(* Logix 5000 project; controller TP_EOL20161211 1769-L16ER-BB1B rev 20.12; software revision 20.01 *)

TASK SocketInterface (periodic, rate 100 ms, priority 2, watchdog 500 ms) : Comm

MODULES
   Local : 1769-L16ER-BB1B (PointIO 0, rev 20.12)
      EOL_ENBT_S02 : 1768-ENBT (Ethernet 192.168.1.20, rev 4.1)
         EOL_PLC_S00 : 1768-L43 (1768Ctrl3Slot 0, rev 20.1)
      Discrete_IO : Embedded (PointIO 1, rev 20.11, Output RPI 20 ms)
END_MODULES

TYPE SKT_Addr :
STRUCT
   Family : INT;   // Address Family Must be 2
   Port : INT;   // Port Number
   Addr : SINT[4];   // IP Address
END_STRUCT
END_TYPE

TYPE SKT_CreateParams :
STRUCT
   Type : DINT;   // 1 - TCP 2- UPD
   Addr : SKT_Addr;
END_STRUCT
END_TYPE

TYPE SKT_DATA_CLIENT :
STRUCT
   MSG_Path : STRING;
   Timeout : DINT;
   Create_Source : SKT_CreateParams;
   Instance : DINT;
   Connect_Source : SKT_OpenConnParam;
   Read_Source : SKT_ReadParams;
   Read_Response : SKT_ReadResponse;
   Write_Source : SKT_WriteParams;
   Write_SizeSent : DINT;
END_STRUCT
END_TYPE

TYPE SKT_OpenConnParam :
STRUCT
   Timeout : DINT;
   DestAddr : STRING;
END_STRUCT
END_TYPE

TYPE SKT_ReadParams :
STRUCT
   Timeout : DINT;
   BufLen : DINT;
END_STRUCT
END_TYPE

TYPE SKT_ReadResponse :
STRUCT
   FromAddr : SKT_Addr;
   Buffer : STR_480;
END_STRUCT
END_TYPE

TYPE SKT_WriteParams :
STRUCT
   Timeout : DINT;
   ToAddr : SKT_Addr;
   Buffer : STR_480;
END_STRUCT
END_TYPE

TYPE STR_480 :
STRUCT
   LEN : DINT;
   DATA : SINT[480];
END_STRUCT
END_TYPE

TYPE UDT_EOLPlus :
STRUCT
   String : STRING[25];
   DINT : DINT[10];
   Real : REAL[10];
END_STRUCT
END_TYPE

ADD_ON_INSTRUCTION SKT_TCP_CLIENT_AOI   (* revision 1.0, ExecutePrescan *)
VAR_IN_OUT
   Client_Data : SKT_DATA_CLIENT; {required}   // This tags holds all the data used by the messages
END_VAR
VAR_INPUT
   Enable_Socket : BOOL; {visible}   // Set by user to enable or disable socket
   Stop_On_Error : BOOL; {visible}   // If any message errors, then delete socket and stop
END_VAR
VAR_IN_OUT
   Create_MSG : MESSAGE; {required}   // Create socket
   Connect_MSG : MESSAGE; {required}   // Connect socket to server.
   Read_MSG : MESSAGE; {required}   // Message to tell socket to return any data it has recieved
   Write_MSG : MESSAGE; {required}   // Write socket message
   Delete_MSG : MESSAGE; {required}   // Delete socket
END_VAR
VAR_OUTPUT
   SC : BOOL; {access Read Only, visible}   // Trying to connect to Server.
   SO : BOOL; {access Read Only, visible}   // Socket connection Open
   DR : BOOL; {access Read Only, visible}   // New Data Ready - Set by AOI when a string is received, cleared by user to acknowledge
   WD : BOOL; {access Read Only, visible}   // Set this bit to Write Data
   ER : BOOL; {access Read Only, visible}   // A message had an ERror
END_VAR
VAR
   State : DINT;   // Current state
END_VAR

ROUTINE Logic   (* ladder *)
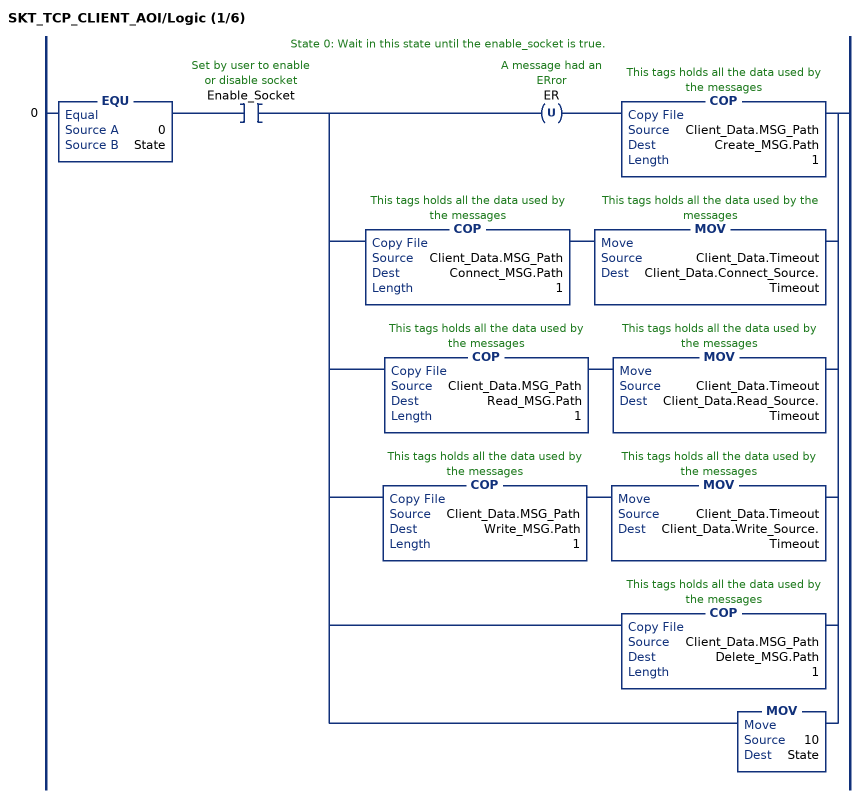
   // State 0: Wait in this state until the enable_socket is true.
   0: EQU(0,State)XIC(Enable_Socket)[OTU(ER) COP(Client_Data.MSG_Path,Create_MSG.Path,1) ,COP(Client_Data.MSG_Path,Connect_MSG.Path,1) MOV(Client_Data.Timeout,Client_Data.Connect_Source.Timeout) ,COP(Client_Data.MSG_Path,Read_MSG.Path,1) MOV(Client_Data.Timeout,Client_Data.Read_Source.Timeout) ,COP(Client_Data.MSG_Path,Write_MSG.Path,1) MOV(Client_Data.Timeout,Client_Data.Write_Source.Timeout) ,COP(Client_Data.MSG_Path,Delete_MSG.Path,1) ,MOV(10,State) ];
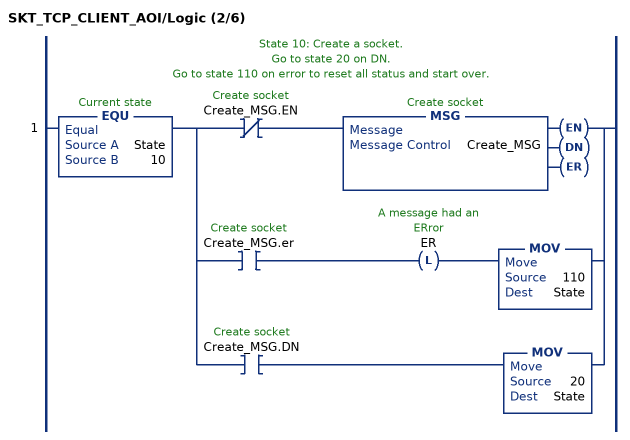
   // State 10: Create a socket.
   // Go to state 20 on DN.
   // Go to state 110 on error to reset all status and start over.
   1: EQU(State,10)[XIO(Create_MSG.EN) MSG(Create_MSG) ,XIC(Create_MSG.er) OTL(ER) MOV(110,State) ,XIC(Create_MSG.DN) MOV(20,State) ];
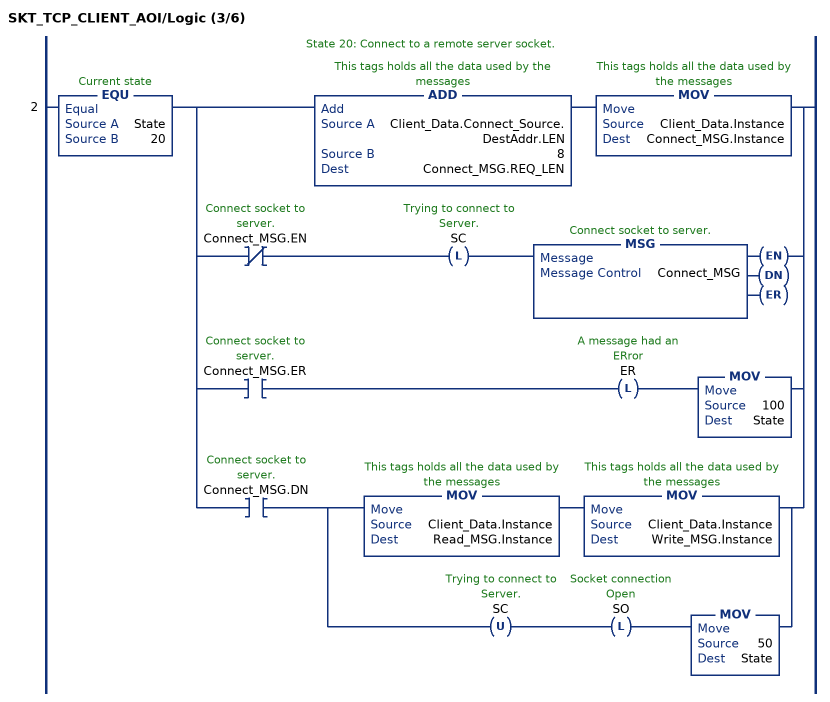
   // State 20: Connect to a remote server socket.
   2: EQU(State,20)[ADD(Client_Data.Connect_Source.DestAddr.LEN,8,Connect_MSG.REQ_LEN) MOV(Client_Data.Instance,Connect_MSG.Instance) ,XIO(Connect_MSG.EN) OTL(SC) MSG(Connect_MSG) ,XIC(Connect_MSG.ER) OTL(ER) MOV(100,State) ,XIC(Connect_MSG.DN) [MOV(Client_Data.Instance,Read_MSG.Instance) MOV(Client_Data.Instance,Write_MSG.Instance) ,OTU(SC) OTL(SO) MOV(50,State) ] ];
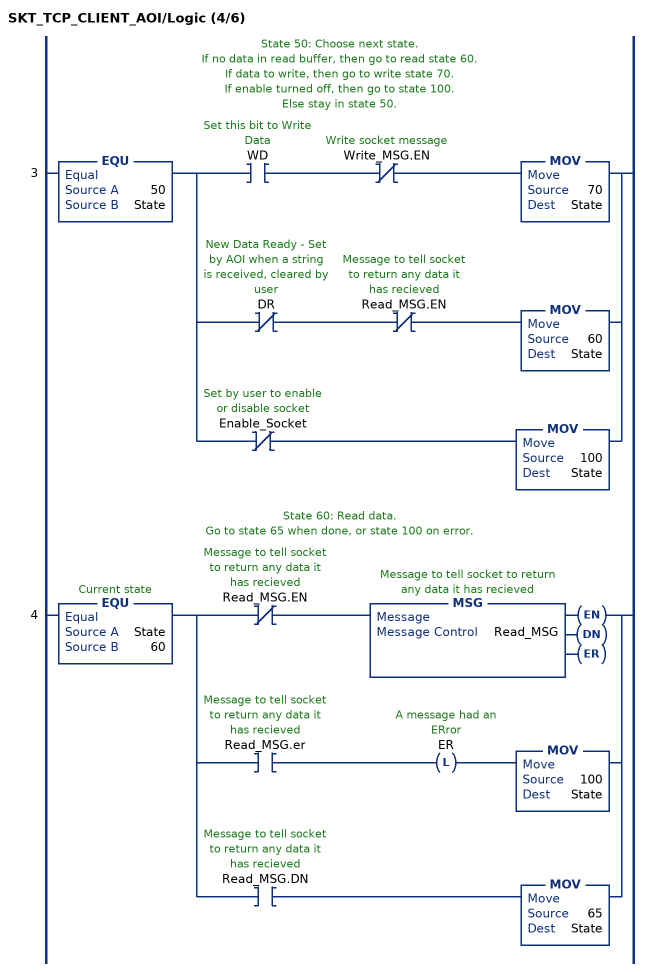
   // State 50: Choose next state.
   // If no data in read buffer, then go to read state 60.
   // If data to write, then go to write state 70.
   // If enable turned off, then go to state 100.
   // Else stay in state 50.
   3: EQU(50,State)[XIC(WD) XIO(Write_MSG.EN) MOV(70,State) ,XIO(DR) XIO(Read_MSG.EN) MOV(60,State) ,XIO(Enable_Socket) MOV(100,State) ];
   // State 60: Read data.
   // Go to state 65 when done, or state 100 on error.
   4: EQU(State,60)[XIO(Read_MSG.EN) MSG(Read_MSG) ,XIC(Read_MSG.er) OTL(ER) MOV(100,State) ,XIC(Read_MSG.DN) MOV(65,State) ];
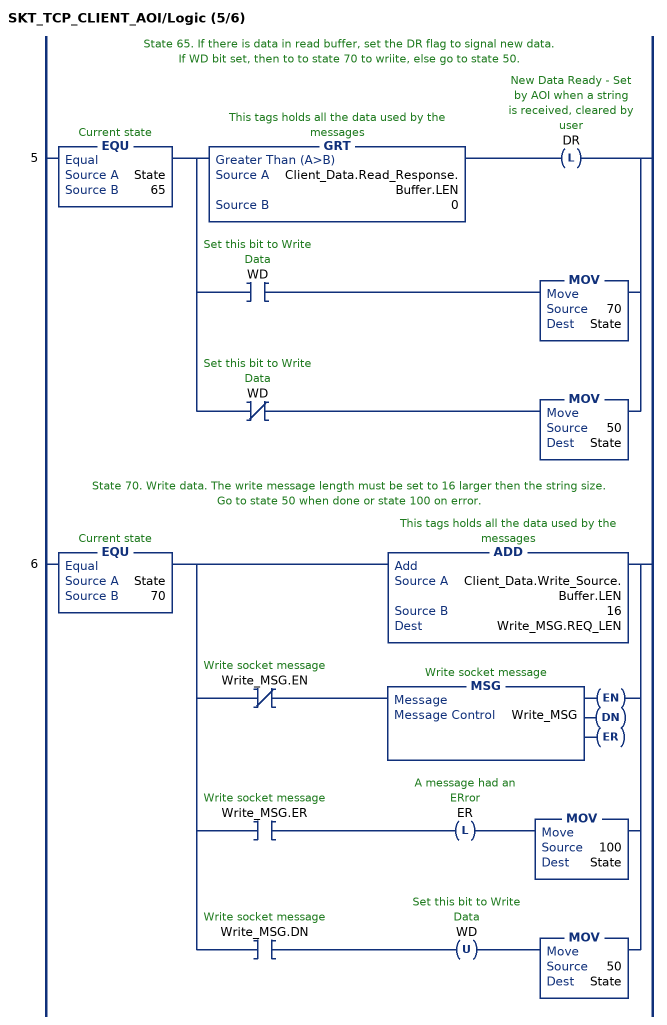
   // State 65. If there is data in read buffer, set the DR flag to signal new data.
   // If WD bit set, then to to state 70 to wriite, else go to state 50.
   5: EQU(State,65)[GRT(Client_Data.Read_Response.Buffer.LEN,0) OTL(DR) ,XIC(WD) MOV(70,State) ,XIO(WD) MOV(50,State) ];
   // State 70. Write data. The write message length must be set to 16 larger then the string size.
   // Go to state 50 when done or state 100 on error.
   6: EQU(State,70)[ADD(Client_Data.Write_Source.Buffer.LEN,16,Write_MSG.REQ_LEN) ,XIO(Write_MSG.EN) MSG(Write_MSG) ,XIC(Write_MSG.ER) OTL(ER) MOV(100,State) ,XIC(Write_MSG.DN) OTU(WD) MOV(50,State) ];
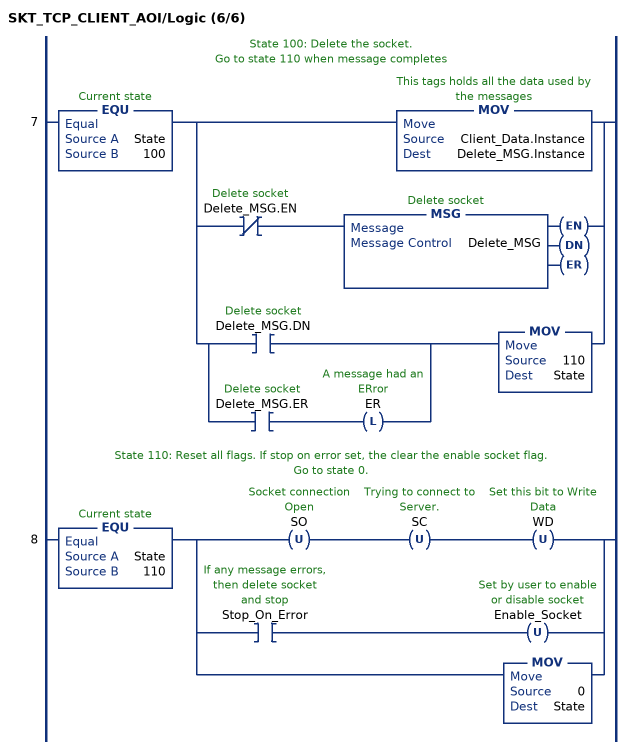
   // State 100: Delete the socket.
   // Go to state 110 when message completes
   7: EQU(State,100)[MOV(Client_Data.Instance,Delete_MSG.Instance) ,XIO(Delete_MSG.EN) MSG(Delete_MSG) ,[XIC(Delete_MSG.DN) ,XIC(Delete_MSG.ER) OTL(ER) ] MOV(110,State) ];
   // State 110: Reset all flags. If stop on error set, the clear the enable socket flag.
   // Go to state 0.
   8: EQU(State,110)[OTU(SO) OTU(SC) OTU(WD) ,XIC(Stop_On_Error) OTU(Enable_Socket) ,MOV(0,State) ];
END_ROUTINE

ROUTINE Prescan   (* ladder *)
// Prescan
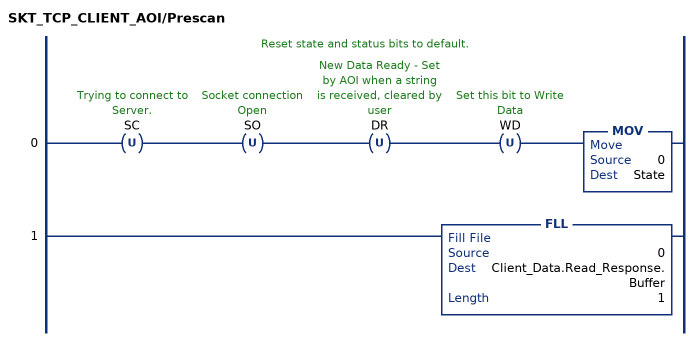
   // Reset state and status bits to default.
   0: OTU(SC)OTU(SO)OTU(DR)OTU(WD)MOV(0,State);
   1: FLL(0,Client_Data.Read_Response.Buffer,1);
END_ROUTINE
END_ADD_ON_INSTRUCTION

VAR_GLOBAL   (* controller tags *)
   ACW_CO_Step : INT;
   ACW_SKT_Client_Connect_MSG : MESSAGE;
        MessageParameters(ServiceCode := 16#004c, LocalElement := ACW_SKT_Client_DATA.Connect_Source, ...)
   ACW_SKT_Client_Create_MSG : MESSAGE;
        MessageParameters(ServiceCode := 16#004b, LocalElement := ACW_SKT_Client_DATA.Create_Source, DestinationTag := ACW_SKT_Client_DATA.Instance, ...)
   ACW_SKT_Client_DATA : SKT_DATA_CLIENT := (MSG_Path := '$01$00', Timeout := 2000, Create_Source.Type := 1, Create_Source.Addr.Family := 2, Instance := 27231, Connect_Source.Timeout := 2000, Connect_Source.DestAddr := '192.168.1.68?port=50001', Read_Source.Timeout := 2000, Read_Source.BufLen := 480, Read_Response.Buffer := '$0233991118247.001$03', Write_Source.Timeout := 2000, Write_Source.ToAddr.Family := 2, Write_Source.Buffer := '$02339$03', Write_SizeSent := 5);
   ACW_SKT_Client_Delete_MSG : MESSAGE;
        MessageParameters(ServiceCode := 16#004f, ...)
   ACW_SKT_Client_Port : DINT;
   ACW_SKT_Client_Read_MSG : MESSAGE;
        MessageParameters(ServiceCode := 16#004d, LocalElement := ACW_SKT_Client_DATA.Read_Source, DestinationTag := ACW_SKT_Client_DATA.Read_Response, ...)
   ACW_SKT_Client_Write_MSG : MESSAGE;
        MessageParameters(ServiceCode := 16#004e, LocalElement := ACW_SKT_Client_DATA.Write_Source, DestinationTag := ACW_SKT_Client_DATA.Write_SizeSent, ...)
   ACW_SKT_Delete_All_MSG : MESSAGE;
        MessageParameters(ServiceCode := 16#0051, ...)
   ACW_SKT_Device_IP_Port_Server : STRING := '192.168.1.68?port=50001';
   ACW_SKT_MSG_PATH : STRING := '$01$00';
   ACW_SKT_String_recieved : STR_480 := '$020100000100$03';
   ACW_SKT_String_to_send : STR_480 := '$02339$03';
   ACW_SKT_Toggle : DINT := -2147482592;
        .0   // Toggle to delete all sockets
   EOL_MSGRead : MESSAGE;
        MessageParameters(ServiceCode := 16#004c, LocalElement := nc_CO_Cmd, ...)
   EOL_MSGWrite : MESSAGE;
        MessageParameters(ServiceCode := 16#004d, LocalElement := np_CO_Status, ...)
   nc_CO_Cmd : UDT_EOLPlus := (String[2] := '5177', String[3] := '457', String[4] := '84', DINT[0] := 2);
   nc_COData : UDT_EOLPlus;
   nc_COData_String : STRING[25];
   np_CO_Status : UDT_EOLPlus := (DINT[0] := 1);
   SKT_Delete_All_MSG : MESSAGE;
        MessageParameters(ServiceCode := 16#0051, ...)
   VDS_SKT_Client_Connect_MSG : MESSAGE;
        MessageParameters(ServiceCode := 16#004c, LocalElement := VDS_SKT_Client_DATA.Connect_Source, ...)
   VDS_SKT_Client_Create_MSG : MESSAGE;
        MessageParameters(ServiceCode := 16#004b, LocalElement := VDS_SKT_Client_DATA.Create_Source, DestinationTag := VDS_SKT_Client_DATA.Instance, ...)
   VDS_SKT_Client_DATA : SKT_DATA_CLIENT := (MSG_Path := '$01$00', Timeout := 2000, Create_Source.Type := 1, Create_Source.Addr.Family := 2, Instance := 19462, Connect_Source.Timeout := 2000, Connect_Source.DestAddr := '192.168.1.66?port=3004', Read_Source.Timeout := 2000, Read_Source.BufLen := 480, Write_Source.Timeout := 2000, Write_Source.ToAddr.Family := 2, Write_Source.Buffer := 'SEL|82254066|$0D', Write_SizeSent := 14);
   VDS_SKT_Client_Delete_MSG : MESSAGE;
        MessageParameters(ServiceCode := 16#004f, ...)
   VDS_SKT_Client_Port : DINT;
   VDS_SKT_Client_Read_MSG : MESSAGE;
        MessageParameters(ServiceCode := 16#004d, LocalElement := VDS_SKT_Client_DATA.Read_Source, DestinationTag := VDS_SKT_Client_DATA.Read_Response, ...)
   VDS_SKT_Client_Write_MSG : MESSAGE;
        MessageParameters(ServiceCode := 16#004e, LocalElement := VDS_SKT_Client_DATA.Write_Source, DestinationTag := VDS_SKT_Client_DATA.Write_SizeSent, ...)
   VDS_SKT_Delete_All_MSG : MESSAGE;
        MessageParameters(ServiceCode := 16#0051, ...)
   VDS_SKT_Device_IP_Port_Server : STRING := '192.168.1.66?port=3004';
   VDS_SKT_MSG_PATH : STRING := '$01$00';
   VDS_SKT_String_recieved : STR_480 := 'ACK$0D';
   VDS_SKT_String_to_send : STR_480 := 'SEL|82254066|$0D';
   VDS_SKT_Toggle : DINT := 1056;
        .0   // Toggle to delete all sockets
   VOS_SKT_Client_Connect_MSG : MESSAGE;
        MessageParameters(ServiceCode := 16#004c, LocalElement := VOS_SKT_Client_DATA.Connect_Source, ...)
   VOS_SKT_Client_Create_MSG : MESSAGE;
        MessageParameters(ServiceCode := 16#004b, LocalElement := VOS_SKT_Client_DATA.Create_Source, DestinationTag := VOS_SKT_Client_DATA.Instance, ...)
   VOS_SKT_Client_DATA : SKT_DATA_CLIENT := (MSG_Path := '$01$00', Timeout := 2000, Create_Source.Type := 1, Create_Source.Addr.Family := 2, Instance := 26707, Connect_Source.Timeout := 2000, Connect_Source.DestAddr := '192.168.1.65?port=3003', Read_Source.Timeout := 2000, Read_Source.BufLen := 480, Write_Source.Timeout := 2000, Write_Source.ToAddr.Family := 2, Write_Source.Buffer := 'SLA|82254066|PLC01=6455B002A4|$0D', Write_SizeSent := 31);
   VOS_SKT_Client_Delete_MSG : MESSAGE;
        MessageParameters(ServiceCode := 16#004f, ...)
   VOS_SKT_Client_Port : DINT;
   VOS_SKT_Client_Read_MSG : MESSAGE;
        MessageParameters(ServiceCode := 16#004d, LocalElement := VOS_SKT_Client_DATA.Read_Source, DestinationTag := VOS_SKT_Client_DATA.Read_Response, ...)
   VOS_SKT_Client_Write_MSG : MESSAGE;
        MessageParameters(ServiceCode := 16#004e, LocalElement := VOS_SKT_Client_DATA.Write_Source, DestinationTag := VOS_SKT_Client_DATA.Write_SizeSent, ...)
   VOS_SKT_Delete_All_MSG : MESSAGE;
        MessageParameters(ServiceCode := 16#0051, ...)
   VOS_SKT_Device_IP_Port_Server : STRING := '192.168.1.65?port=3003';
   VOS_SKT_MSG_PATH : STRING := '$01$00';
   VOS_SKT_String_recieved : STR_480 := 'JDL|6|Copy of Field00=82254066|Copy of Field02=HAIR FALL CONTROL|Copy of Field04=10:06|Copy of Field03=14902430400883|Copy of Field01=|PLC01=6455B002A4|$0D';
   VOS_SKT_String_to_send : STR_480 := 'GJN$0D';
   VOS_SKT_Toggle : DINT := 1056;
        .0   // Toggle to delete all sockets
   wrk_Ons : INT := 512;
END_VAR

PROGRAM Comm   (* main routine Main *)
VAR
   aa_Dint : DINT := 2;
   aa_FSC : CONTROL := (LEN := 20, POS := 9, EN := 1, IN := 1, FD := 1);
   aa_STD : CONTROL := (LEN := 20);
   aa_STD1 : CONTROL := (LEN := 6);
   ACW_Add : DINT;
   ACW_Cmd_ConvStart : BOOL;
   ACW_Cmd_ConvStop : BOOL := 1;
   ACW_CO_Timer : TIMER[10] := ([0].PRE := 1000);
   acw_ConvStopped : STRING := '$020100000100$03';
   ACW_SKT_Client_AOI : SKT_TCP_CLIENT_AOI := (Enable_Socket := 1, SO := 1, DR := 1);
   Araa : CONTROL := (LEN := 20, POS := 17);
   Array : REAL[20] := ([6] := 2.0, [7] := 15.0, [8] := 45.0, [9] := 54.0, [10] := 54.0, [11] := 55.0, [12] := 55.0, [13] := 55.3, [14] := 56.0, [15] := 56.2, [16] := 56.5, [17] := 57.0, [18] := 57.8, [19] := 65.0);
   Array2 : REAL[20];
   Cmd_ACW_ConvStart : STRING := '$0212$03'; {constant}
   Cmd_ACW_ConvStop : STRING := '$02339$03'; {constant}
   Cmd_ACW_RecipeName : STRING := '91118247.001';
   Cmd_ACW_RecipeNumber : STRING := '$0220001$03';
   Cmd_ACW_SetRecipeName : BOOL;
   Cmd_ACW_SetRecipeNumber : BOOL;
   Cmd_ACW_SetTargetLL : BOOL;
   Cmd_ACW_SetTargetUL : BOOL;
   Cmd_ACW_SetTargetWeight : BOOL;
   Cmd_ACW_Status : STRING;
   Cmd_ACW_TargetLL : STRING := '84';
   Cmd_ACW_TargetUL : STRING := '457';
   Cmd_ACW_TargetWeight : STRING := '5177';
   Cmd_Chk : INT;
   Cmd_RecipeNo : BOOL;
   Cmd_RequestData : STRING := '$020$03'; {constant}
   Cmd_VJDS_GJD : BOOL;
   Cmd_VJDS_GJF : BOOL;
   Cmd_VJDS_GJN : BOOL;
   Cmd_VJDS_GST : BOOL;
   Cmd_VJDS_OfflineRequest : BOOL;
   Cmd_VJDS_RunRequest : BOOL;
   Cmd_VJDS_SEL : BOOL;
   Cmd_VJDS_ShutDownRequest : BOOL;
   Cmd_VJDS_ShuttingDownRequest : BOOL;
   Cmd_VJDS_SLA : BOOL;
   Cmd_VJDS_StartupRequest : BOOL;
   Cmd_VJOS_GJD : BOOL;
   Cmd_VJOS_GJF : BOOL;
   Cmd_VJOS_GJN : BOOL;
   Cmd_VJOS_GST : BOOL;
   Cmd_VJOS_OfflineRequest : BOOL;
   Cmd_VJOS_RunRequest : BOOL;
   Cmd_VJOS_ShutDownRequest : BOOL;
   Cmd_VJOS_ShuttingDownRequest : BOOL;
   Cmd_VJOS_SLA : BOOL;
   Cmd_VJOS_StartupRequest : BOOL;
   CO_Complete : TIMER := (PRE := 180000);
   CO_Trigger : DINT := 6;
   CO_VJCTU : COUNTER := (ACC := 2, CU := 1, DN := 1);
   CO_VJCTUOS : COUNTER := (ACC := 2, CU := 1, DN := 1);
   FSC : CONTROL;
   Par_JobSelect : STRING := '82254066';
   Par_RecipeName : STRING := '$02239$03';
   Par_TargetLL : STRING := '$02203-$03';
   Par_TargetUL : STRING := '$02202$03';
   Par_TargetWeight : STRING := '$02201$03';
   Par_VarData : STRING := '6455B002A4';
   Par_VJ_JobSelect : STRING := '82254066';
   RCO_Triggered : INT := 4;
   Real_STD : REAL := 27.257544;
   Sts_Conv : STRING := '1';
   Sts_VJDS_CurrentJob : STRING;
   Sts_VJOS_CurrentJob : STRING := '82254066';
   VDS_SKT_Client_AOI : SKT_TCP_CLIENT_AOI := (Enable_Socket := 1, SO := 1);
   VJ_ACK : STRING := 'ACK$0D';
   VJ_Blank : STRING;
   VJ_FieldData : STRING := '6455B002A4';
   VJ_FieldDataDS : STRING;
   VJ_FieldPos : INT := 136;
   VJ_FieldPosDS : INT;
   VJ_PLC01 : STRING := 'PLC01='; {constant}
   VJ_VarDataPOS : INT := 142;
   VJDS_JobFieldDataErr : BOOL;
   VJDS_JobFieldDataNA : BOOL;
   VJDS_JobSLAErr : BOOL;
   VJDS_msgSeq : INT := 60;
   VJDS_ReadTimer : TIMER[10] := ([0].PRE := 2000, [1].PRE := 2000, [2].PRE := 2000, [3].PRE := 2000, [3].ACC := 2000, [3].EN := 1, [3].DN := 1, [4].PRE := 2000, [5].PRE := 2000, [6].PRE := 3000);
   VJDS_Wrk_Jobassign : STRING := '82254066|PLC01=6455B002A4';
   VJDS_wrk_ONS : DINT;
   VJOS_JobFieldDataErr : BOOL;
   VJOS_JobSLAErr : BOOL;
   VJOS_msgSeq : INT := 30;
   VJOS_ReadTimer : TIMER[10] := ([0].PRE := 2000, [1].PRE := 2000, [2].PRE := 2000, [2].ACC := 2000, [2].EN := 1, [2].DN := 1, [3].PRE := 2000, [4].PRE := 2000, [5].PRE := 2000, [6].PRE := 3000);
   VJOS_Seq : INT := 10;
   VJOS_Wrk_Jobassign : STRING := '82254066|PLC01=6455B002A4';
   VJOS_wrk_ONS : DINT := 32;
   VOS_SKT_Client_AOI : SKT_TCP_CLIENT_AOI := (Enable_Socket := 1, SO := 1);
   wrk_Concat : STRING := '82254066|PLC01=';
   wrk_ConcatSLA : STRING := '|PLC01='; {constant}
   wrk_GJD : STRING := 'GJD$0D'; {constant}
   wrk_GJF : STRING := 'GJF||$0D'; {constant}
   wrk_GJN : STRING := 'GJN$0D'; {constant}
   wrk_GST : STRING := 'GST$0D'; {constant}
   wrk_SEL : STRING := 'SEL||$0D'; {constant}
   wrk_SLA : STRING := 'SLA||$0D'; {constant}
   wrk_State : STRING := '3';
   wrk_StateCmd : STRING := 'SST||$0D'; {constant}
END_VAR

ROUTINE Anritsu   (* ladder *)
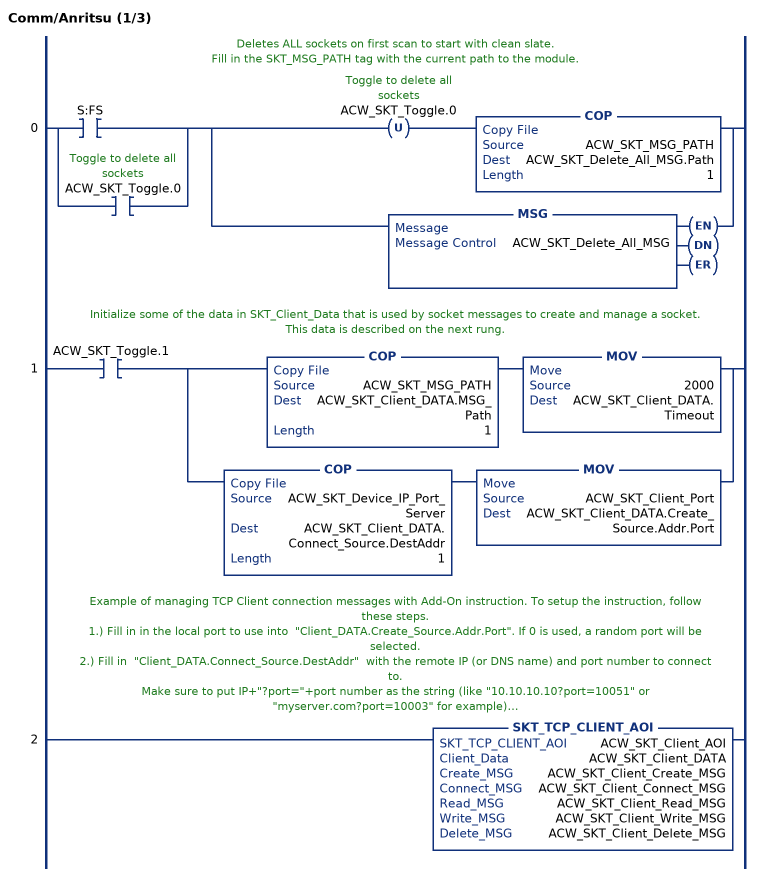
   // Deletes ALL sockets on first scan to start with clean slate.
   // Fill in the SKT_MSG_PATH tag with the current path to the module.
   0: [XIC(S:FS) ,XIC(ACW_SKT_Toggle.0) ][OTU(ACW_SKT_Toggle.0) COP(ACW_SKT_MSG_PATH,ACW_SKT_Delete_All_MSG.Path,1) ,MSG(ACW_SKT_Delete_All_MSG) ];
   // Initialize some of the data in SKT_Client_Data that is used by socket messages to create and manage a socket.
   // This data is described on the next rung.
   1: XIC(ACW_SKT_Toggle.1)[COP(ACW_SKT_MSG_PATH,ACW_SKT_Client_DATA.MSG_Path,1) MOV(2000,ACW_SKT_Client_DATA.Timeout) ,COP(ACW_SKT_Device_IP_Port_Server,ACW_SKT_Client_DATA.Connect_Source.DestAddr,1) MOV(ACW_SKT_Client_Port,ACW_SKT_Client_DATA.Create_Source.Addr.Port) ];
   // Example of managing TCP Client connection messages with Add-On instruction. To setup the instruction, follow these steps.
   // 1.) Fill in in the local port to use into  "Client_DATA.Create_Source.Addr.Port". If 0 is used, a random port will be selected.
   // 2.) Fill in  "Client_DATA.Connect_Source.DestAddr"  with the remote IP (or DNS name) and port number to connect to.
   // Make sure to put IP+"?port="+port number as the string (like "10.10.10.10?port=10051" or "myserver.com?port=10003" for example).
   // 3.) Fill in the path to the module in the SKT_MSG_PATH tag (the path will look like "$01$03" for slot 3, for example).
   // 4.) To start or stop the client connection, set or clear the Enable_Socket respectively.
   // 5.) If trying to trap error for troubleshooting the connection, the set the Stop_on_Error bit on the instruction. If there is an error, the instruction will clear the Stop_on_Errorwhen a message errors.
   // The SC status bit means trying to connect. The SO status bit means Socket Connected and open. The ER bit means a message ERrored.
   // When the DR bit is set by the instruction, then there is string data that arrived from the socket. Copy the string data if desired and clear the DR bit to get new data.
   // When data needs to be sent by the application, fill in the string data into "Client_DATA.Write_Source.Buffer", then set the WD bit. The instruction will clear the WD bit when the data is written.
   // Modify the rung branches to suit the application.
   2: SKT_TCP_CLIENT_AOI(ACW_SKT_Client_AOI,ACW_SKT_Client_DATA,ACW_SKT_Client_Create_MSG,ACW_SKT_Client_Connect_MSG,ACW_SKT_Client_Read_MSG,ACW_SKT_Client_Write_MSG,ACW_SKT_Client_Delete_MSG);
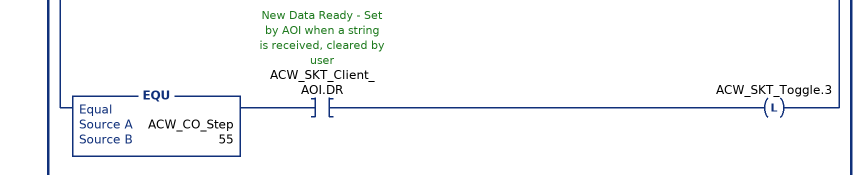
   3: [EQU(ACW_CO_Step,0) [XIC(ACW_Cmd_ConvStart) ONS(wrk_Ons.8) COP(Cmd_ACW_ConvStart,ACW_SKT_String_to_send,Cmd_ACW_ConvStart.LEN) ,XIC(ACW_Cmd_ConvStop) ONS(wrk_Ons.9) COP(Cmd_ACW_ConvStop,ACW_SKT_String_to_send,Cmd_ACW_ConvStop.LEN) ] OTL(ACW_SKT_Toggle.2) ,XIC(nc_CO_Cmd.DINT[0].2) ONS(wrk_Ons.1) MOV(10,ACW_CO_Step) ,XIO(ACW_CO_Timer[0].DN) LIM(10,ACW_CO_Step,60) TON(ACW_CO_Timer[0],?,?) ,XIC(ACW_CO_Timer[0].DN) ADD(ACW_CO_Step,5,ACW_CO_Step) ,EQU(ACW_CO_Step,10) XIO(ACW_SKT_Client_AOI.WD) COP(Cmd_ACW_RecipeNumber,ACW_SKT_String_to_send,Cmd_ACW_RecipeNumber.LEN) OTL(ACW_SKT_Toggle.2) ,EQU(ACW_CO_Step,15) XIC(ACW_SKT_Client_AOI.DR) OTL(ACW_SKT_Toggle.3) ,EQU(ACW_CO_Step,20) XIO(ACW_SKT_Client_AOI.WD) INSERT(Par_RecipeName,Cmd_ACW_RecipeName,5,ACW_SKT_String_to_send) OTL(ACW_SKT_Toggle.2) ,EQU(ACW_CO_Step,25) XIC(ACW_SKT_Client_AOI.DR) OTL(ACW_SKT_Toggle.3) ,EQU(ACW_CO_Step,30) XIO(ACW_SKT_Client_AOI.WD) INSERT(Par_TargetWeight,Cmd_ACW_TargetWeight,5,ACW_SKT_String_to_send) OTL(ACW_SKT_Toggle.2) ,EQU(ACW_CO_Step,35) XIC(ACW_SKT_Client_AOI.DR) OTL(ACW_SKT_Toggle.3) ,EQU(ACW_CO_Step,40) XIO(ACW_SKT_Client_AOI.WD) INSERT(Par_TargetUL,Cmd_ACW_TargetUL,5,ACW_SKT_String_to_send) OTL(ACW_SKT_Toggle.2) ,EQU(ACW_CO_Step,45) XIC(ACW_SKT_Client_AOI.DR) OTL(ACW_SKT_Toggle.3) ,EQU(ACW_CO_Step,50) XIO(ACW_SKT_Client_AOI.WD) INSERT(Par_TargetLL,Cmd_ACW_TargetLL,6,ACW_SKT_String_to_send) OTL(ACW_SKT_Toggle.2) ,EQU(ACW_CO_Step,55) XIC(ACW_SKT_Client_AOI.DR) OTL(ACW_SKT_Toggle.3) ];
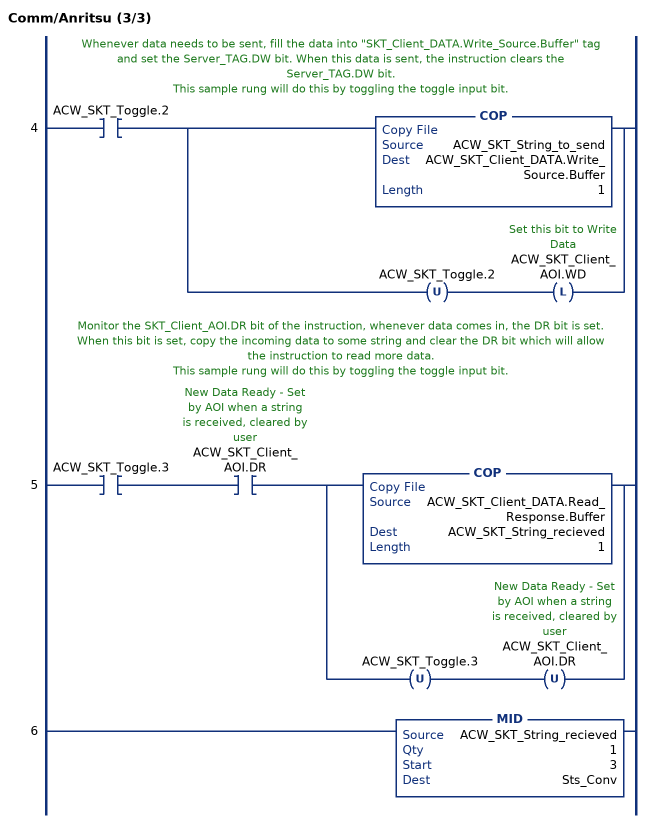
   // Whenever data needs to be sent, fill the data into "SKT_Client_DATA.Write_Source.Buffer" tag and set the Server_TAG.DW bit. When this data is sent, the instruction clears the Server_TAG.DW bit.
   // This sample rung will do this by toggling the toggle input bit.
   4: XIC(ACW_SKT_Toggle.2)[COP(ACW_SKT_String_to_send,ACW_SKT_Client_DATA.Write_Source.Buffer,1) ,OTU(ACW_SKT_Toggle.2) OTL(ACW_SKT_Client_AOI.WD) ];
   // Monitor the SKT_Client_AOI.DR bit of the instruction, whenever data comes in, the DR bit is set. When this bit is set, copy the incoming data to some string and clear the DR bit which will allow the instruction to read more data.
   // This sample rung will do this by toggling the toggle input bit.
   5: XIC(ACW_SKT_Toggle.3)XIC(ACW_SKT_Client_AOI.DR)[COP(ACW_SKT_Client_DATA.Read_Response.Buffer,ACW_SKT_String_recieved,1) ,OTU(ACW_SKT_Toggle.3) OTU(ACW_SKT_Client_AOI.DR) ];
   6: MID(ACW_SKT_String_recieved,1,3,Sts_Conv);
END_ROUTINE

ROUTINE Main   (* ladder *)
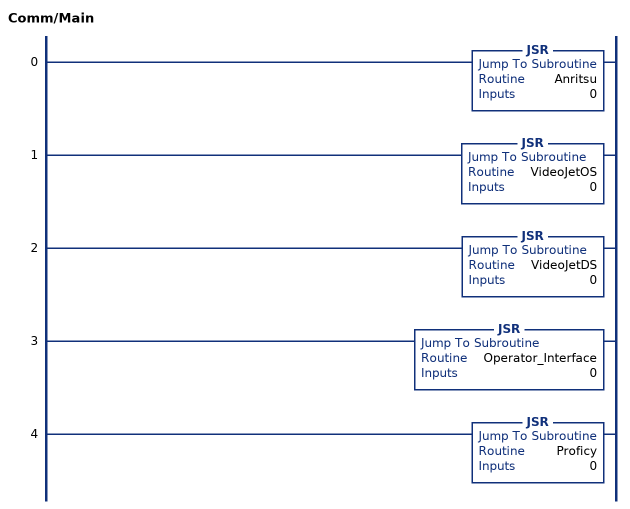
   0: JSR(Anritsu,0);
   1: JSR(VideoJetOS,0);
   2: JSR(VideoJetDS,0);
   3: JSR(Operator_Interface,0);
   4: JSR(Proficy,0);
END_ROUTINE

ROUTINE Operator_Interface   (* ladder *)
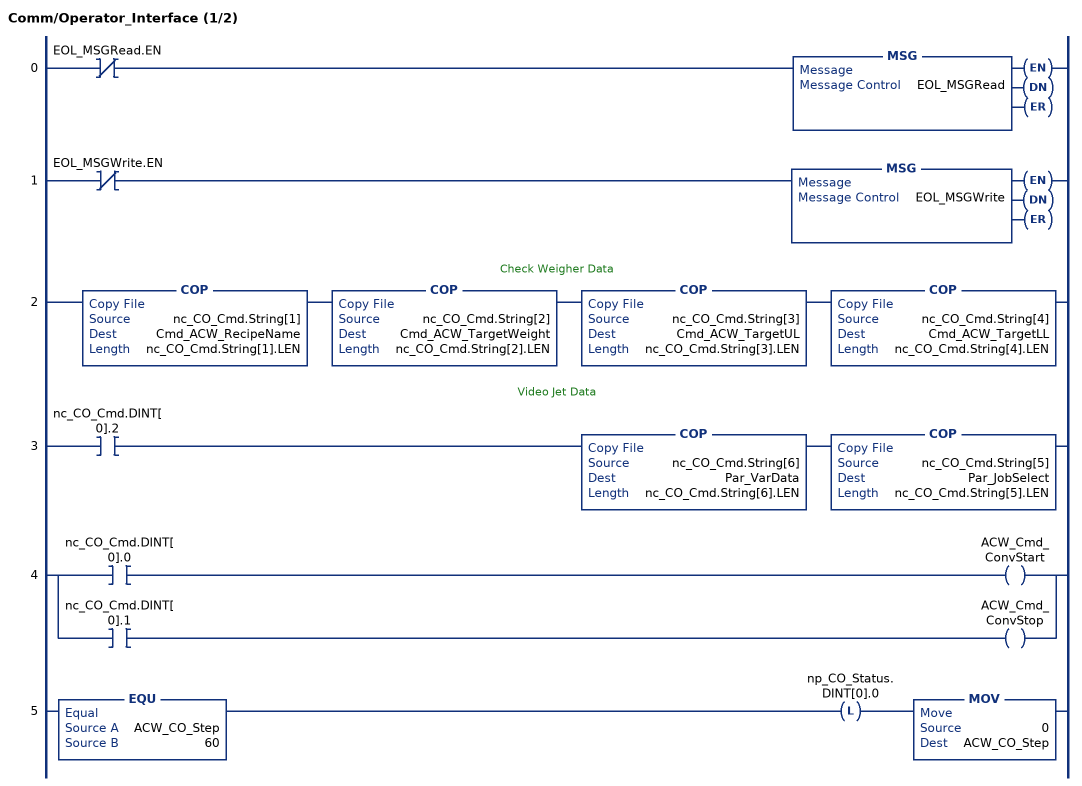
   0: XIO(EOL_MSGRead.EN)MSG(EOL_MSGRead);
   1: XIO(EOL_MSGWrite.EN)MSG(EOL_MSGWrite);
   // Check Weigher Data
   2: COP(nc_CO_Cmd.String[1],Cmd_ACW_RecipeName,nc_CO_Cmd.String[1].LEN)COP(nc_CO_Cmd.String[2],Cmd_ACW_TargetWeight,nc_CO_Cmd.String[2].LEN)COP(nc_CO_Cmd.String[3],Cmd_ACW_TargetUL,nc_CO_Cmd.String[3].LEN)COP(nc_CO_Cmd.String[4],Cmd_ACW_TargetLL,nc_CO_Cmd.String[4].LEN);
   // Video Jet Data
   3: XIC(nc_CO_Cmd.DINT[0].2)COP(nc_CO_Cmd.String[6],Par_VarData,nc_CO_Cmd.String[6].LEN)COP(nc_CO_Cmd.String[5],Par_JobSelect,nc_CO_Cmd.String[5].LEN);
   4: [XIC(nc_CO_Cmd.DINT[0].0) OTE(ACW_Cmd_ConvStart) ,XIC(nc_CO_Cmd.DINT[0].1) OTE(ACW_Cmd_ConvStop) ];
   5: EQU(ACW_CO_Step,60)OTL(np_CO_Status.DINT[0].0)MOV(0,ACW_CO_Step);
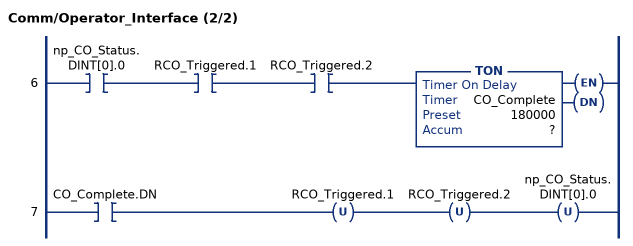
   6: XIC(np_CO_Status.DINT[0].0)XIC(RCO_Triggered.1)XIC(RCO_Triggered.2)TON(CO_Complete,?,?);
   7: XIC(CO_Complete.DN)OTU(RCO_Triggered.1)OTU(RCO_Triggered.2)OTU(np_CO_Status.DINT[0].0);
END_ROUTINE

ROUTINE Proficy   (* ladder *)
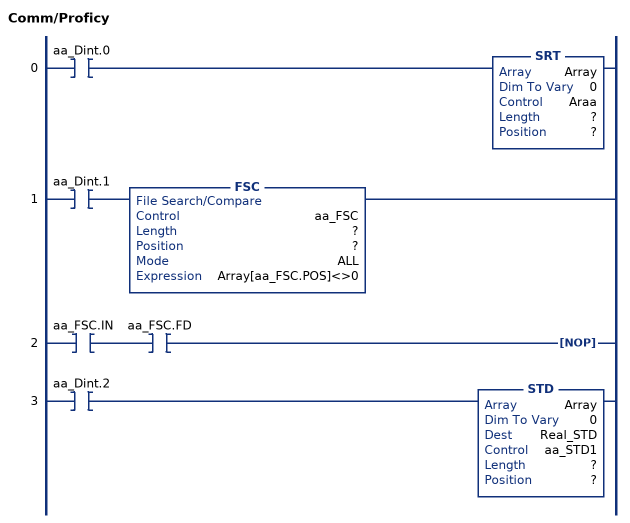
   0: XIC(aa_Dint.0)SRT(Array,0,Araa,?,?);
   1: XIC(aa_Dint.1)FSC(aa_FSC,?,?,ALL,Array[aa_FSC.POS]<>0);
   2: XIC(aa_FSC.IN)XIC(aa_FSC.FD)NOP();
   3: XIC(aa_Dint.2)STD(Array,0,Real_STD,aa_STD1,?,?);
END_ROUTINE

ROUTINE VideoJetDS   (* ladder *)
// 192.168.1.66
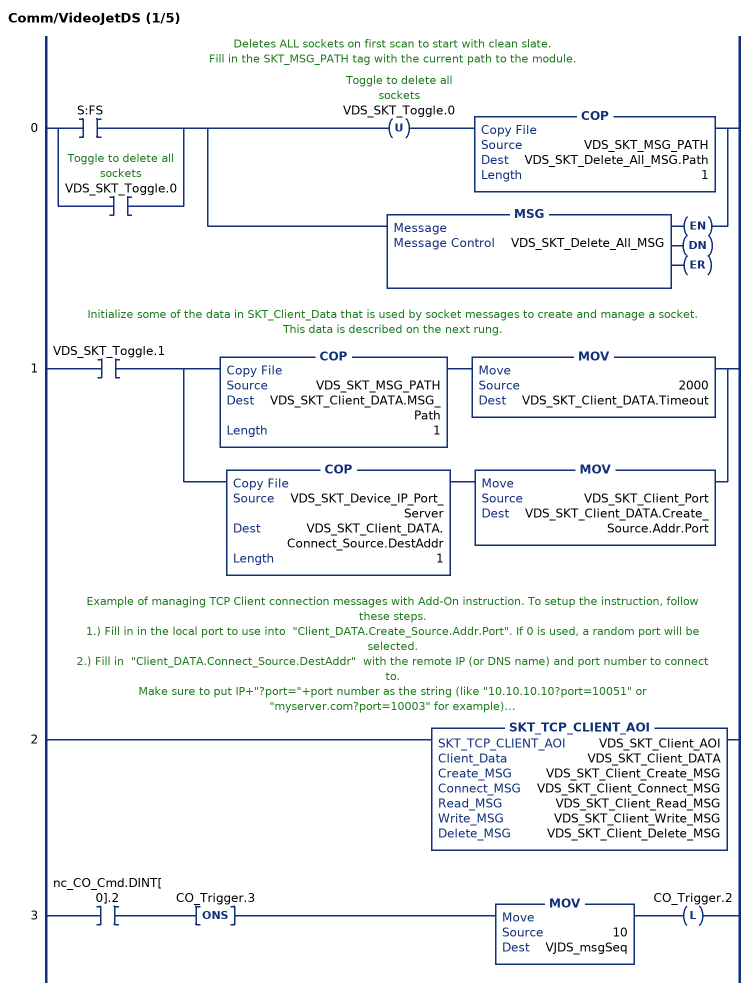
   // Deletes ALL sockets on first scan to start with clean slate.
   // Fill in the SKT_MSG_PATH tag with the current path to the module.
   0: [XIC(S:FS) ,XIC(VDS_SKT_Toggle.0) ][OTU(VDS_SKT_Toggle.0) COP(VDS_SKT_MSG_PATH,VDS_SKT_Delete_All_MSG.Path,1) ,MSG(VDS_SKT_Delete_All_MSG) ];
   // Initialize some of the data in SKT_Client_Data that is used by socket messages to create and manage a socket.
   // This data is described on the next rung.
   1: XIC(VDS_SKT_Toggle.1)[COP(VDS_SKT_MSG_PATH,VDS_SKT_Client_DATA.MSG_Path,1) MOV(2000,VDS_SKT_Client_DATA.Timeout) ,COP(VDS_SKT_Device_IP_Port_Server,VDS_SKT_Client_DATA.Connect_Source.DestAddr,1) MOV(VDS_SKT_Client_Port,VDS_SKT_Client_DATA.Create_Source.Addr.Port) ];
   // Example of managing TCP Client connection messages with Add-On instruction. To setup the instruction, follow these steps.
   // 1.) Fill in in the local port to use into  "Client_DATA.Create_Source.Addr.Port". If 0 is used, a random port will be selected.
   // 2.) Fill in  "Client_DATA.Connect_Source.DestAddr"  with the remote IP (or DNS name) and port number to connect to.
   // Make sure to put IP+"?port="+port number as the string (like "10.10.10.10?port=10051" or "myserver.com?port=10003" for example).
   // 3.) Fill in the path to the module in the SKT_MSG_PATH tag (the path will look like "$01$03" for slot 3, for example).
   // 4.) To start or stop the client connection, set or clear the Enable_Socket respectively.
   // 5.) If trying to trap error for troubleshooting the connection, the set the Stop_on_Error bit on the instruction. If there is an error, the instruction will clear the Stop_on_Errorwhen a message errors.
   // The SC status bit means trying to connect. The SO status bit means Socket Connected and open. The ER bit means a message ERrored.
   // When the DR bit is set by the instruction, then there is string data that arrived from the socket. Copy the string data if desired and clear the DR bit to get new data.
   // When data needs to be sent by the application, fill in the string data into "Client_DATA.Write_Source.Buffer", then set the WD bit. The instruction will clear the WD bit when the data is written.
   // Modify the rung branches to suit the application.
   2: SKT_TCP_CLIENT_AOI(VDS_SKT_Client_AOI,VDS_SKT_Client_DATA,VDS_SKT_Client_Create_MSG,VDS_SKT_Client_Connect_MSG,VDS_SKT_Client_Read_MSG,VDS_SKT_Client_Write_MSG,VDS_SKT_Client_Delete_MSG);
   3: XIC(nc_CO_Cmd.DINT[0].2)ONS(CO_Trigger.3)MOV(10,VJDS_msgSeq)OTL(CO_Trigger.2);
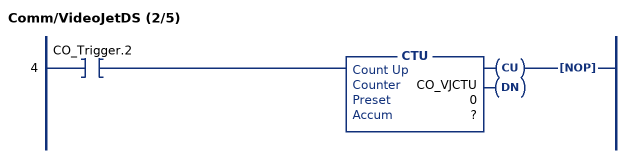
   4: XIC(CO_Trigger.2)CTU(CO_VJCTU,?,?)NOP();
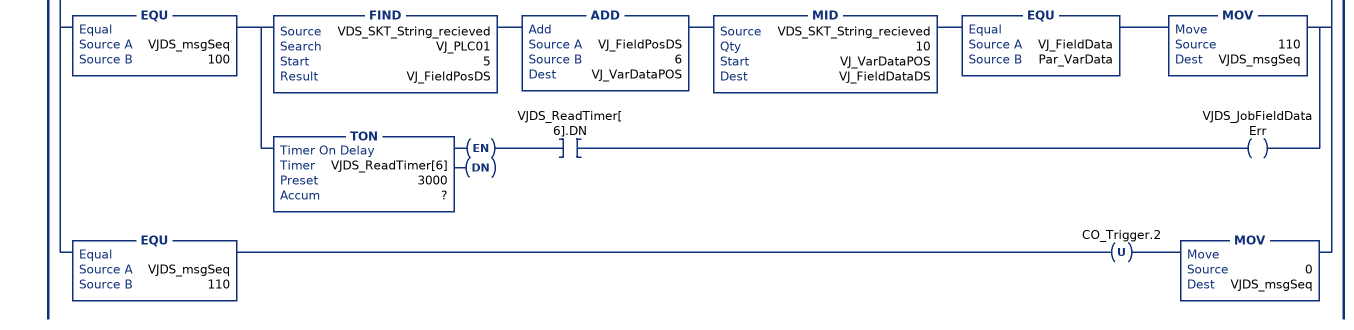
   5: [EQU(VJDS_msgSeq,10) [XIC(VDS_SKT_Client_AOI.DR) TON(VJDS_ReadTimer[0],?,?) XIC(VJDS_ReadTimer[0].DN) OTL(VDS_SKT_Toggle.3) ,XIO(VDS_SKT_Client_AOI.DR) TON(VJDS_ReadTimer[1],?,?) XIC(VJDS_ReadTimer[1].DN) MOV(20,VJDS_msgSeq) ] ,EQU(VJDS_msgSeq,20) NEQ(VJ_Blank,Par_VJ_JobSelect) [NEQ(VJ_Blank,Par_VarData) ,XIO(VJDS_JobFieldDataNA) ] OTL(Cmd_VJDS_SLA) MOV(25,VJDS_msgSeq) ,EQU(VJDS_msgSeq,25) OTL(VDS_SKT_Toggle.2) XIC(VDS_SKT_Client_AOI.WD) MOV(30,VJDS_msgSeq) ,EQU(VJDS_msgSeq,30) TON(VJDS_ReadTimer[2],?,?) XIC(VJDS_ReadTimer[2].DN) XIC(VDS_SKT_Client_AOI.DR) OTL(VDS_SKT_Toggle.3) MOV(40,VJDS_msgSeq) ,EQU(VJDS_msgSeq,40) EQU(VJ_ACK,VDS_SKT_String_recieved) OTL(VDS_SKT_Toggle.3) MOV(50,VJDS_msgSeq) ,EQU(VJDS_msgSeq,50) OTL(Cmd_VJDS_GJN) MOV(55,VJDS_msgSeq) ,EQU(VJDS_msgSeq,55) OTL(VDS_SKT_Toggle.2) XIC(VDS_SKT_Client_AOI.WD) MOV(60,VJDS_msgSeq) ,EQU(VJDS_msgSeq,60) TON(VJDS_ReadTimer[3],?,?) XIC(VJDS_ReadTimer[3].DN) XIC(VDS_SKT_Client_AOI.DR) OTL(VDS_SKT_Toggle.3) MOV(70,VJDS_msgSeq) ,EQU(VJDS_msgSeq,70) [MID(VDS_SKT_String_recieved,8,5,Sts_VJDS_CurrentJob) EQU(Sts_VJDS_CurrentJob,Par_VJ_JobSelect) MOV(80,VJDS_msgSeq) ,TON(VJDS_ReadTimer[5],?,?) XIC(VJDS_ReadTimer[5].DN) OTE(VJDS_JobSLAErr) ] ,EQU(VJDS_msgSeq,80) [XIC(VJDS_JobFieldDataNA) OTL(Cmd_VJDS_GJD) MOV(85,VJDS_msgSeq) ,XIO(VJDS_JobFieldDataNA) MOV(110,VJDS_msgSeq) ] ,EQU(VJDS_msgSeq,85) OTL(VDS_SKT_Toggle.2) XIC(VDS_SKT_Client_AOI.WD) MOV(90,VJDS_msgSeq) ,EQU(VJDS_msgSeq,90) TON(VJDS_ReadTimer[4],?,?) XIC(VJDS_ReadTimer[4].DN) XIC(VDS_SKT_Client_AOI.DR) OTL(VDS_SKT_Toggle.3) MOV(100,VJDS_msgSeq) ,EQU(VJDS_msgSeq,100) [FIND(VDS_SKT_String_recieved,VJ_PLC01,5,VJ_FieldPosDS) ADD(VJ_FieldPosDS,6,VJ_VarDataPOS) MID(VDS_SKT_String_recieved,10,VJ_VarDataPOS,VJ_FieldDataDS) EQU(VJ_FieldData,Par_VarData) MOV(110,VJDS_msgSeq) ,TON(VJDS_ReadTimer[6],?,?) XIC(VJDS_ReadTimer[6].DN) OTE(VJDS_JobFieldDataErr) ] ,EQU(VJDS_msgSeq,110) OTU(CO_Trigger.2) MOV(0,VJDS_msgSeq) ];
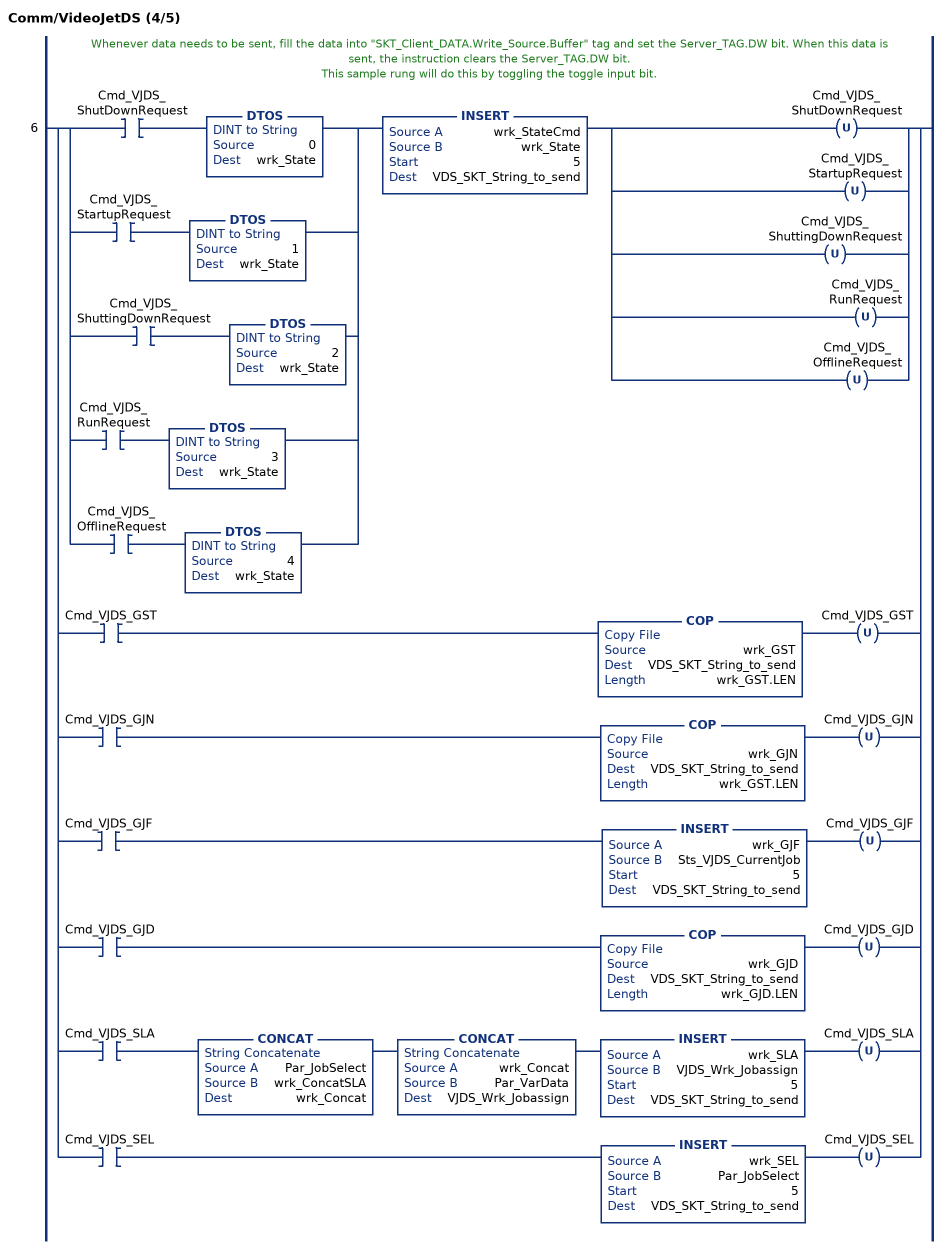
   // Whenever data needs to be sent, fill the data into "SKT_Client_DATA.Write_Source.Buffer" tag and set the Server_TAG.DW bit. When this data is sent, the instruction clears the Server_TAG.DW bit.
   // This sample rung will do this by toggling the toggle input bit.
   6: [[XIC(Cmd_VJDS_ShutDownRequest) DTOS(0,wrk_State) ,XIC(Cmd_VJDS_StartupRequest) DTOS(1,wrk_State) ,XIC(Cmd_VJDS_ShuttingDownRequest) DTOS(2,wrk_State) ,XIC(Cmd_VJDS_RunRequest) DTOS(3,wrk_State) ,XIC(Cmd_VJDS_OfflineRequest) DTOS(4,wrk_State) ] INSERT(wrk_StateCmd,wrk_State,5,VDS_SKT_String_to_send) [OTU(Cmd_VJDS_ShutDownRequest) ,OTU(Cmd_VJDS_StartupRequest) ,OTU(Cmd_VJDS_ShuttingDownRequest) ,OTU(Cmd_VJDS_RunRequest) ,OTU(Cmd_VJDS_OfflineRequest) ] ,XIC(Cmd_VJDS_GST) COP(wrk_GST,VDS_SKT_String_to_send,wrk_GST.LEN) OTU(Cmd_VJDS_GST) ,XIC(Cmd_VJDS_GJN) COP(wrk_GJN,VDS_SKT_String_to_send,wrk_GST.LEN) OTU(Cmd_VJDS_GJN) ,XIC(Cmd_VJDS_GJF) INSERT(wrk_GJF,Sts_VJDS_CurrentJob,5,VDS_SKT_String_to_send) OTU(Cmd_VJDS_GJF) ,XIC(Cmd_VJDS_GJD) COP(wrk_GJD,VDS_SKT_String_to_send,wrk_GJD.LEN) OTU(Cmd_VJDS_GJD) ,XIC(Cmd_VJDS_SLA) CONCAT(Par_JobSelect,wrk_ConcatSLA,wrk_Concat) CONCAT(wrk_Concat,Par_VarData,VJDS_Wrk_Jobassign) INSERT(wrk_SLA,VJDS_Wrk_Jobassign,5,VDS_SKT_String_to_send) OTU(Cmd_VJDS_SLA) ,XIC(Cmd_VJDS_SEL) INSERT(wrk_SEL,Par_JobSelect,5,VDS_SKT_String_to_send) OTU(Cmd_VJDS_SEL) ];
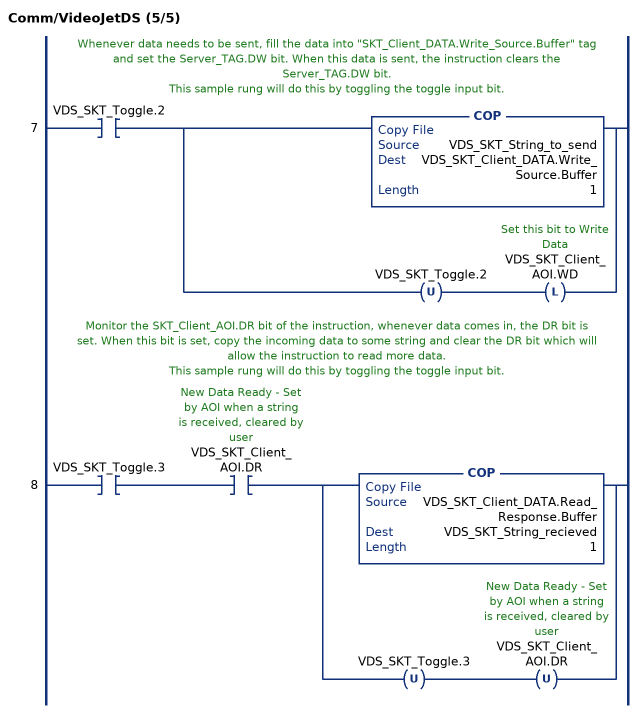
   // Whenever data needs to be sent, fill the data into "SKT_Client_DATA.Write_Source.Buffer" tag and set the Server_TAG.DW bit. When this data is sent, the instruction clears the Server_TAG.DW bit.
   // This sample rung will do this by toggling the toggle input bit.
   7: XIC(VDS_SKT_Toggle.2)[COP(VDS_SKT_String_to_send,VDS_SKT_Client_DATA.Write_Source.Buffer,1) ,OTU(VDS_SKT_Toggle.2) OTL(VDS_SKT_Client_AOI.WD) ];
   // Monitor the SKT_Client_AOI.DR bit of the instruction, whenever data comes in, the DR bit is set. When this bit is set, copy the incoming data to some string and clear the DR bit which will allow the instruction to read more data.
   // This sample rung will do this by toggling the toggle input bit.
   8: XIC(VDS_SKT_Toggle.3)XIC(VDS_SKT_Client_AOI.DR)[COP(VDS_SKT_Client_DATA.Read_Response.Buffer,VDS_SKT_String_recieved,1) ,OTU(VDS_SKT_Toggle.3) OTU(VDS_SKT_Client_AOI.DR) ];
END_ROUTINE
